// TIA Portal V19 export
VAR_GLOBAL   // PLC tag table "NEW AI"
   "LT-1" AT %IW176 : Int;
   "CT-1" AT %IW178 : Int;
   "CT-2" AT %IW180 : Int;
   "LT-2" AT %IW182 : Int;
   "AI-5 SPARE1" AT %IW184 : Int;
   "AI-6 SPARE2" AT %IW186 : Int;
   "AI-7 SPARE3" AT %IW188 : Int;
   "AI-8 SPARE4" AT %IW190 : Int;
END_VAR
